FUNCTION TN_prod : real
VAR
	i:DINT;
END_VAR
VAR_IN_OUT
	Inputs: ARRAY[*] OF REAL;
END_VAR

TN_prod:=1;
FOR i:=LOWER_BOUND(Inputs,1) TO UPPER_BOUND(Inputs,1) DO
	TN_prod:=TN_prod*inputs[i];
END_FOR

END_FUNCTION

(* stored: Version 1.1.0.1, ProductVersion 3.1.4024.6
   POU TN_prod: Id {c2a72472-2f27-47a1-a627-cfda9d6c2e03}, SpecialFunc None *)
